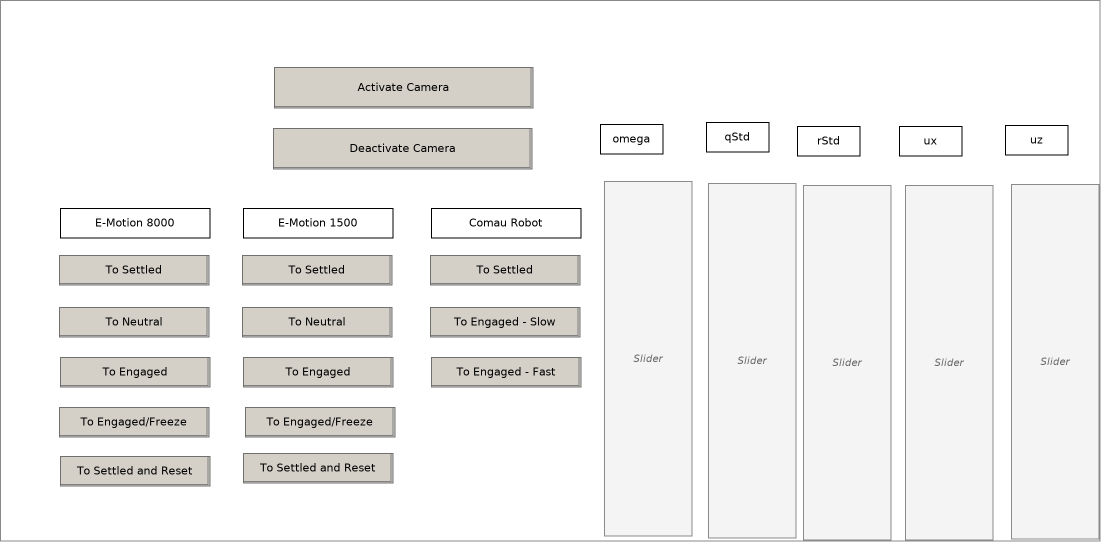
VISUALIZATION HMI  // 1101x542
    Button (430,255 150x30), "To Settled"
        OnMouseClick: execute { MotionLab.COMAU.Control.mode := 0; }
    Rectangle (431,208 150x30), "Comau Robot"
    Button (430,307 150x30), "To Engaged - Slow"
        OnMouseClick: execute { MotionLab.COMAU.Control.mode := 1; }
    Button (431,357 150x30), "To Engaged - Fast"
        OnMouseClick: execute { MotionLab.COMAU.Control.mode := 2; }
    Slider (604,181 88x355), variable: MotionLab.COMAU.Control.omega, scale 1..100
    Rectangle (600,124 63x30), "omega"
    Button (242,255 150x30), "To Settled"
        OnMouseClick: execute { MotionLab.EM1500.Control.CMND := 1; }
    Rectangle (243,208 150x30), "E-Motion 1500"
    Button (242,307 150x30), "To Neutral"
        OnMouseClick: execute { MotionLab.EM1500.Control.CMND := 3; }
    Button (243,357 150x30), "To Engaged"
        OnMouseClick: execute { MotionLab.EM1500.Control.CMND := 7; }
    Button (243,453 150x30), "To Settled and Reset"
        OnMouseClick: execute { MotionLab.EM1500.Control.CMND := 17; }
    Button (59,255 150x30), "To Settled"
        OnMouseClick: execute { MotionLab.EM8000.Control.CMND := 1; }
    Rectangle (60,208 150x30), "E-Motion 8000"
    Button (59,307 150x30), "To Neutral"
        OnMouseClick: execute { MotionLab.EM8000.Control.CMND := 3; }
    Button (60,357 150x30), "To Engaged"
        OnMouseClick: execute { MotionLab.EM8000.Control.CMND := 7; }
    Button (60,456 150x30), "To Settled and Reset"
        OnMouseClick: execute { MotionLab.EM8000.Control.CMND := 17; }
    Button (59,407 150x30), "To Engaged/Freeze"
        OnMouseClick: execute { MotionLab.EM8000.Control.CMND := 15; }
    Button (245,407 150x30), "To Engaged/Freeze"
        OnMouseClick: execute { MotionLab.EM1500.Control.CMND := 15; }
    Slider (708,183 88x355), variable: MotionLab.qStd, scale 0.1..10
    Rectangle (706,122 63x30), "qStd"
    Slider (803,185 88x355), variable: MotionLab.rStd, scale 0.1..20
    Rectangle (797,126 63x30), "rStd"
    Button (274,67 259x41), "Activate Camera"
        OnMouseClick: execute { MotionLab.camActive := TRUE; }
    Button (273,128 259x41), "Deactivate Camera"
        OnMouseClick: execute { MotionLab.camActive := FALSE; }
    Slider (905,185 88x355), variable: MotionLab.getPose.ux, scale 0.3..1.2
    Rectangle (899,126 63x30), "ux"
    Slider (1011,184 88x355), variable: MotionLab.getPose.uz, scale -2..-1.5
    Rectangle (1005,125 63x30), "uz"
END_VISUALIZATION

(* stored: Version 1.1.0.1, ProductVersion 3.1.4020.6
   Visu HMI: Id {bcd56803-f2f0-499c-ae2a-7c6913391d84} *)
